(* Logix 5000 project; controller Machine_Maintenance_Lab2 vendor 1 type 14 code 155 rev 36.11; software revision 36.00 *)

TASK MainTask (continuous, watchdog 500 ms) : MainProgram

MODULES
   Local : vendor 1 type 14 code 155 (PointIO 0, rev 36.11)
      Discrete_IO : Embedded (PointIO 1, rev 36.11, Output RPI 20 ms)
END_MODULES

PROGRAM MainProgram   (* main routine MainRoutine *)
VAR
   Arm_OneShot : BOOL;
   ArmCount : COUNTER := (PRE := 1);
   counter : COUNTER := (PRE := 5);
   CycleCounter : COUNTER := (PRE := 5);
   delay : TIMER := (PRE := 50);
   HighCycleTimer : COUNTER := (PRE := 700);
   i_ArmDown : ALIAS FOR Local:1:I.Data.3;
   i_CycleDone : ALIAS FOR o_CycleDone;
   i_GreenPB : ALIAS FOR Local:1:I.Data.0;
   i_GreenPB_ConveyorStart : ALIAS FOR i_GreenPB;
   i_GreenPBLight_Conveyor1ON : ALIAS FOR o_GreenPBLight_Conveyor1ON;
   i_Pause : ALIAS FOR Pause;
   i_Piston : ALIAS FOR Local:1:O.Data.2;
   i_RedPB_StopButton : ALIAS FOR Local:1:I.Data.1;
   i_RedPBLight_Conveyor2ON : ALIAS FOR o_RedPBLight_Conveyor2ON;
   i_Turnkey : ALIAS FOR Local:1:I.Data.2;
   i_Turnkey_ItemSensor : ALIAS FOR i_Turnkey;
   ItemCounter1 : COUNTER := (PRE := 5);
   ItemCounterLeft : COUNTER := (PRE := 5);
   ItemCounterRight : COUNTER := (PRE := 6);
   LowCycleTimer : COUNTER := (PRE := 300);
   NewCycle : BOOL;
   o_CycleDone : BOOL;
   o_GreenPBLight : ALIAS FOR Local:1:O.Data.0;
   o_GreenPBLight_Conveyor1ON : ALIAS FOR o_GreenPBLight;
   o_Piston : ALIAS FOR i_Piston;
   o_RedPBLight : ALIAS FOR Local:1:O.Data.1;
   o_RedPBLight_Conveyor2ON : ALIAS FOR o_RedPBLight;
   o_YellowLight : ALIAS FOR Local:1:O.Data.2;
   OS_Out : BOOL;
   Pause : BOOL;
   PrintDone : BOOL;
   PrinterArmTime : TIMER := (PRE := 1000);
   ResetDelay : TIMER := (PRE := 500);
   SheetDetectReset : COUNTER := (PRE := 1);
   ThreeSecTimer : TIMER := (PRE := 3000);
   timer : TIMER := (PRE := 5000);
   TimerHighCycle : TIMER := (PRE := 700);
   TimerLowCycle : TIMER := (PRE := 300);
   Travel_StampTime : TIMER := (PRE := 2000);
   TurnkeyOneShot : BOOL;
END_VAR

ROUTINE MainRoutine   (* ladder *)
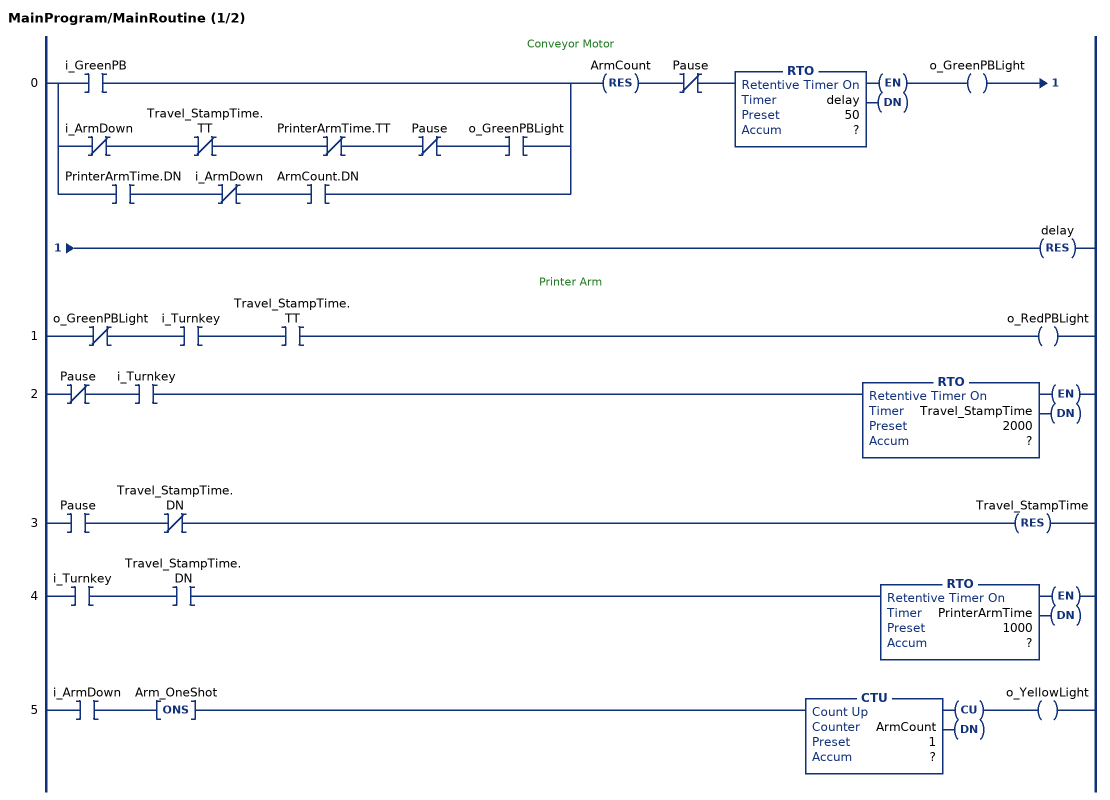
   // Conveyor Motor
   0: [XIC(i_GreenPB) ,[XIO(i_ArmDown) XIO(Travel_StampTime.TT) XIO(PrinterArmTime.TT) XIO(Pause) XIC(o_GreenPBLight) ,XIC(PrinterArmTime.DN) XIO(i_ArmDown) XIC(ArmCount.DN) ] ]RES(ArmCount)XIO(Pause)RTO(delay,?,?)OTE(o_GreenPBLight)RES(delay);
   // Printer Arm
   1: XIO(o_GreenPBLight)XIC(i_Turnkey)XIC(Travel_StampTime.TT)OTE(o_RedPBLight);
   2: XIO(Pause)XIC(i_Turnkey)RTO(Travel_StampTime,?,?);
   3: XIC(Pause)XIO(Travel_StampTime.DN)RES(Travel_StampTime);
   4: XIC(i_Turnkey)XIC(Travel_StampTime.DN)RTO(PrinterArmTime,?,?);
   5: XIC(i_ArmDown)ONS(Arm_OneShot)CTU(ArmCount,?,?)OTE(o_YellowLight);
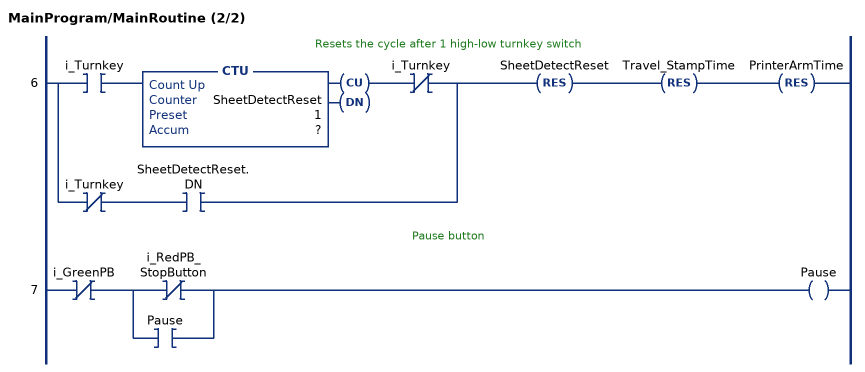
   // Resets the cycle after 1 high-low turnkey switch
   6: [XIC(i_Turnkey) CTU(SheetDetectReset,?,?) XIO(i_Turnkey) ,XIO(i_Turnkey) XIC(SheetDetectReset.DN) ]RES(SheetDetectReset)RES(Travel_StampTime)RES(PrinterArmTime);
   // Pause button
   7: XIO(i_GreenPB)[XIO(i_RedPB_StopButton) ,XIC(Pause) ]OTE(Pause);
END_ROUTINE
END_PROGRAM
